# EPICS autosave request: iocBoot/ioc13laser_ultra/auto_positions.req
file "CARS_motor_positions.req",       P=$(P), M=m1
~
